INTERFACE ITF_GroupE_TE2_HMI_Init EXTENDS ITF_BaseGroupElement, ITF_GroupE_TE2_HMI_Connector

END_INTERFACE

(* stored: Version 1.1.0.1, ProductVersion 3.1.4024.15
   Itf ITF_GroupE_TE2_HMI_Init: Id {4e4f7d85-847d-49f1-9ce4-22091056cc97} *)
